// TIA Portal project "Reaktor2_Wizualizacja" (V17)

(* hardware
DEVICE "S7-1500/ET200MP station_1"  S7-1500 station
   slot 0: "Rail_0"  Rack  6ES7 590-1***0-0AA0
   slot 1: "PLC_1"  CPU 1512C-1 PN  6ES7 512-1CK00-0AB0  V2.9
      slot 3: "CPU display_1"  6ES7591-1AA00-0AA0
      slot 32768: "PROFINET interface_1"  X1
         slot 32769: "Port_1"  X1 P1
         slot 32770: "Port_2"  X1 P2
      slot 34817: "Virtual CP interface port_1"  Virtual CP interface port  Virtual CP interface port
DEVICE "PC_System_1"  SIMATIC PC station
   slot 0: "SIMATIC PC station"  Rail  SIMATIC PC-Station  V1.0
      slot 125: "Stationmanager"  Station_Manager  V6.0.4
   slot 1: "HMI_RT_1"  WinCC RT Professional  6AV2 105-0xxxx-xxxx  17.0.0.0
   slot 2: "IE general_1"  IE General  IE_CP  V8.2.0
      slot 1: "PROFINET interface"  IEGeneral.Interface.8.2.0
*)

// ===== PLC "PLC_1"  CPU 1512C-1 PN =====

VAR_GLOBAL   // PLC tag table "Default tag table"
   "System_Byte" AT %MB1 : Byte;
   "FirstScan" AT %M1.0 : Bool;
   "DiagStatusUpdate" AT %M1.1 : Bool;
   "AlwaysTRUE" AT %M1.2 : Bool;
   "AlwaysFALSE" AT %M1.3 : Bool;
   "Clock_Byte" AT %MB0 : Byte;
   "Clock_10Hz" AT %M0.0 : Bool;
   "Clock_5Hz" AT %M0.1 : Bool;
   "Clock_2.5Hz" AT %M0.2 : Bool;
   "Clock_2Hz" AT %M0.3 : Bool;
   "Clock_1.25Hz" AT %M0.4 : Bool;
   "Clock_1Hz" AT %M0.5 : Bool;
   "Clock_0.625Hz" AT %M0.6 : Bool;
   "Clock_0.5Hz" AT %M0.7 : Bool;
   "iAktualny_poziom" AT %MD8 : Real;   // czujnik pomiaru aktualnego poziomu czynników znajdujących się w reaktorze
   "iAktualna_temperatura" AT %MD12 : Real;   // czujnik pomiaru aktualnej wartości temperatury czynników znajdujących się w reaktorze
   "iWartość_zadana_poziomu" AT %MD16 : Real;   // AI3 - wartość zadana poziomu
   "iWartość_zadana_temperatury" AT %MD20 : Real;   // AI4 - wartość zadana temperatury
END_VAR

VAR_GLOBAL   // PLC tag table "zmienne_z_modułów"
   "xNapełnianie_reaktora" AT %M2.0 : Bool;   // Faza Napełnianie reaktora
   "xPodgrzewanie_produktu" AT %M2.1 : Bool;   // Faza Podgrzewanie produktu w reaktorze
   "xChłodzenie_reaktora" AT %M2.2 : Bool;   // Faza Chłodzenie produktu
   "xOpróżnianie_reaktora" AT %M2.3 : Bool;   // Faza Opróżnianie reaktora
   "xPraca_Man/Auto" AT %M2.4 : Bool;   // Przełącznik pracy Man/Auto
   "xZawór_V1" AT %M3.0 : Bool;   // zawór V1 - doprowadzenie czynnika A (oznaczenie V1)
   "xZawór_V2" AT %M3.1 : Bool;   // zawór V2 - doprowadzenie czynnika B (oznaczenie V2)
   "xZawór_V3" AT %M3.2 : Bool;   // Dopływ medium chłodzącego (oznaczenie V3)
   "xZawór_V4" AT %M3.3 : Bool;   // Odpływ medium chłodzącego (oznaczenie V4)
   "xZawór_V5" AT %M3.4 : Bool;   // V5 - Odpływ medium ogrzewającego (oznaczenie V5)
   "xSilnik_M" AT %M3.5 : Bool;   // M - Mieszadło wprawiane w ruch przez silnik (oznaczenie M)
   "iZawór_AV1" AT %MW4 : Int;   // Odprowadzenie produktu końcowego (oznaczenie AV1)
   "iZawór_AV2" AT %MW6 : Int;   // AV2 - Dopływ medium ogrzewającego (oznaczenie AV2)
END_VAR

DATA_BLOCK "Napełnianie_reaktora_DB"   // DB1
{ S7_Optimized_Access := 'FALSE' }
VERSION : 0.1
// stored: InstanceOfName Napełnianie_reaktora
"Napełnianie_reaktora"
BEGIN
END_DATA_BLOCK

DATA_BLOCK "Podgrzewanie_produktu_w_reaktorze_DB"   // DB2
{ S7_Optimized_Access := 'FALSE' }
VERSION : 0.1
// stored: InstanceOfName Podgrzewanie_produktu_w_reaktorze
"Podgrzewanie_produktu_w_reaktorze"
BEGIN
END_DATA_BLOCK

DATA_BLOCK "Chłodzenie_produktu_DB"   // DB3
{ S7_Optimized_Access := 'FALSE' }
VERSION : 0.1
// stored: InstanceOfName Chłodzenie_produktu
"Chłodzenie_produktu"
BEGIN
END_DATA_BLOCK

DATA_BLOCK "Opróżnianie_reaktora_DB"   // DB4
{ S7_Optimized_Access := 'FALSE' }
VERSION : 0.1
// stored: InstanceOfName Opróżnianie_reaktora
"Opróżnianie_reaktora"
BEGIN
END_DATA_BLOCK

DATA_BLOCK "zmienne_OB1"   // DB5
{ S7_Optimized_Access := 'FALSE' }
VERSION : 0.1
   VAR
      uiWybór_fazy_reaktora : UInt;
      iTemperatura_przed_podgrzaniem : Int;
      iNapełnianie_zbiornika_zakonczone : Int;
      iPodgrzewanie_produktu_zakończone : Int;
      iChłodzenie_reaktora_zakończone : Int;
      iOpróżnianie_reaktora_zakończone : Int;
      xAwaria : Bool;
      xZbocze_narastające_Napełnianie_zbiornika : Bool;
      xZbocze_narastające_Podgrzewanie_produktu : Bool;
      xZbocze_narastające_Chłodzenie_reaktora : Bool;
      xZbocze_narastające_Opróżnianie_reaktora : Bool;
   END_VAR
BEGIN
END_DATA_BLOCK

DATA_BLOCK "Użytkownicy"   // DB6
{ S7_Optimized_Access := 'TRUE' }
VERSION : 0.1
   VAR
      User_name : String;
   END_VAR
BEGIN
END_DATA_BLOCK

DATA_BLOCK "Symulator_grzanie_DB"   // DB8
{ S7_Optimized_Access := 'TRUE' }
VERSION : 0.1
// stored: InstanceOfName Symulator_grzanie
"Symulator_grzanie"
BEGIN
END_DATA_BLOCK

DATA_BLOCK "Symulator_napelniania_DB"   // DB11
{ S7_Optimized_Access := 'TRUE' }
VERSION : 0.1
// stored: InstanceOfName Symulator_napelniania
"Symulator_napelniania"
BEGIN
END_DATA_BLOCK

FUNCTION_BLOCK "Napełnianie_reaktora"   // FB1, SCL
{ S7_Optimized_Access := 'FALSE' }
VERSION : 0.1
   VAR_INPUT
      iAktualny_poziom_w_reaktorze : Real;
      iZadany_poziom : Real;
      iOpróżnianie_reaktora_zakończone : Int;
      xAwaria_lokal : Bool;
   END_VAR
   VAR_OUTPUT
      xZawór_V1 : Bool;   // zawór V1 - doprowadzenie czynnika A (oznaczenie V1)
      xZawór_V2 : Bool;   // zawór V2 - doprowadzenie czynnika B (oznaczenie V2)
      iNapełnianie_zbiornika_zakonczone : Int;
      iZawór_AV1 : Int;
   END_VAR
BEGIN
   ///zabezpiecznie że poprzednia faza opróżniania się zakończyła oraz nie wystąpiła awaria//////
   IF #xAwaria_lokal=0  THEN
       #iNapełnianie_zbiornika_zakonczone := 0;
       //napełnianie czynnikiem A do 1/3 poziomu zadanego otwarcie zaworu V1
       IF (#iAktualny_poziom_w_reaktorze >= 0.9 AND #iAktualny_poziom_w_reaktorze <= (#iZadany_poziom / 3.0)) THEN

           #xZawór_V1 := 1;

       END_IF;

       //po osiągnięciu 1/3 wartości zadanej zamknięcie zaworu V1, otwarcie zaworu V2
       IF (#iAktualny_poziom_w_reaktorze > (#iZadany_poziom / 3.0)) AND (#iAktualny_poziom_w_reaktorze <= #iZadany_poziom) THEN
           #xZawór_V1 := 0;
           #xZawór_V2 := 1;
       END_IF;

       //po osiągnięciu wartości zadanej zamknięcie zaworu V2
       IF (#iAktualny_poziom_w_reaktorze > #iZadany_poziom) THEN
           #xZawór_V2 := 0;
       END_IF;
       IF (#iAktualny_poziom_w_reaktorze > #iZadany_poziom) AND #xZawór_V2 = 0  THEN
           #iNapełnianie_zbiornika_zakonczone := 1;///informacja o zakończeniu fazy napełniania/////
       END_IF;
   END_IF;
   //wystąpienie awarii////
   IF #xAwaria_lokal=1 THEN
       ///zamknięcie zaworów V1, V2////
       #xZawór_V1 := 0;
       #xZawór_V2 := 0;
       ///otwarcie zaworu AV1 do opróżniania zbiornika/////
       IF #iAktualny_poziom_w_reaktorze > 0.0 THEN
           #iZawór_AV1 := 27648;

       END_IF;
       ///zamknięcie zaworu AV1 po opróżnieniu zbiornika////
       IF #iAktualny_poziom_w_reaktorze = 0.0 THEN
           #iZawór_AV1 := 0;
           #iNapełnianie_zbiornika_zakonczone := -1;///informacja o wystąpieniu awarii podczas napełniania////
       END_IF;

   END_IF;
END_FUNCTION_BLOCK

FUNCTION_BLOCK "Podgrzewanie_produktu_w_reaktorze"   // FB2, SCL
{ S7_Optimized_Access := 'FALSE' }
VERSION : 0.1
   VAR_INPUT
      iWartość_zadana_temperatury : Real;
      iAktualna_temperatura : Real;
      iNapełnianie_zbiornika_zakończone : Int;
      iAktualny_poziom_w_reaktorze : Real;
      xAwaria_lokalna : Bool;
   END_VAR
   VAR_OUTPUT
      xOdpływ_medium_ogrzewającego : Bool;
      xMieszadło : Bool;
      iDopływ_medium_ogrzewającego : Int;
      iTemperatura_przed_podgrzaniem : Real;
      iPodgrzewanie_produktu_zakończone : Int;
      iZawór_AV1 : Int;
   END_VAR
   VAR
      iI : Int := 0;
      iK : UInt := 0;
      iCzas_zamykania_zaworu_AV2 : UInt := 10;
      rWartość_zadana_temperatury : Real;
      rAktualna_temperatura : Real;
      rDopływ_medium_ogrzewającego : Real;
      xZbocze_narastające_1Hz : Bool;
   END_VAR
   VAR_TEMP
      "xStart_timera_zamykania zaworu" : Bool;
   END_VAR
BEGIN
   ///zabezpiecznie że poprzednia faza napełniania się zakończyła oraz nie wystąpiła awaria////// 
   IF #iNapełnianie_zbiornika_zakończone=1 AND #xAwaria_lokalna=0 THEN
       #iPodgrzewanie_produktu_zakończone := 0;


       //konwersja typów z INT na REAL
       #rAktualna_temperatura := INT_TO_REAL(#iAktualna_temperatura);
       #rWartość_zadana_temperatury := INT_TO_REAL(#iWartość_zadana_temperatury);

       //przepisanie temperatury produktu przed grzaniem
       WHILE #xOdpływ_medium_ogrzewającego = 0 AND #iI = 0 AND #rDopływ_medium_ogrzewającego <= 0.0 DO
           #iTemperatura_przed_podgrzaniem := #iAktualna_temperatura;
           #iI := #iI + 1;
           //Załączenie mieszadła 
           #xMieszadło := 1;
       END_WHILE;


       //otwarcie zaworu V5 odpływ medium ogrzewającego
       IF #xOdpływ_medium_ogrzewającego = 0 AND #iI = 1 THEN
           #xOdpływ_medium_ogrzewającego := 1;
       END_IF;

       //podgrzewanie produktu do 75% temperatury zadanej otwarcie zaworu AV2 - dopływ medium ogrzewającego
       IF (#rAktualna_temperatura <= (#rWartość_zadana_temperatury * 0.75)) AND (#xOdpływ_medium_ogrzewającego = 1) THEN
           #iDopływ_medium_ogrzewającego := 27648;
       END_IF;


       //po osiągnięciu 75% tempratury zadanej inicjalizacja zamkykania zaworu AV2 - dopływ medium ogrzewającego
       #rDopływ_medium_ogrzewającego := INT_TO_REAL(#iDopływ_medium_ogrzewającego);
       IF #rAktualna_temperatura >= (#rWartość_zadana_temperatury * 0.75) THEN

           #iDopływ_medium_ogrzewającego := 13500;

       END_IF;

       IF #rAktualna_temperatura >= #rWartość_zadana_temperatury THEN
           #iDopływ_medium_ogrzewającego := 0;
       END_IF;


           IF #iDopływ_medium_ogrzewającego<=0 THEN
               //Wyłącznie mieszadła
               #xMieszadło := 0;
               //zamknięcie zaworu V5 odpływ medium ogrzewającego
               #xOdpływ_medium_ogrzewającego := 0;
               #iPodgrzewanie_produktu_zakończone := 1;///informacja o zakończeniu fazy podgrzewania/////
           END_IF;

       END_IF;


   //wystąpienie awarii////
   IF #xAwaria_lokalna=1 THEN
       ///zamknięcie zaworów medium ogrzewającego oraz wyłączenie mieszadła////
       #iDopływ_medium_ogrzewającego := 0;
       #xOdpływ_medium_ogrzewającego := 0;
       #xMieszadło := 0;
       ///otwarcie zaworu AV1 do opróżniania zbiornika/////
       IF #iAktualny_poziom_w_reaktorze > 0.0 THEN
           #iZawór_AV1 := 27648;

       END_IF;
       ///zamknięcie zaworu AV1 po opróżnieniu zbiornika////
       IF #iAktualny_poziom_w_reaktorze = 0.0 THEN
           #iZawór_AV1 := 0;
           #iPodgrzewanie_produktu_zakończone := -1;///informacja o wystąpieniu awarii podczas fazy podgrzewania////
       END_IF;


   END_IF;
END_FUNCTION_BLOCK

FUNCTION_BLOCK "Chłodzenie_produktu"   // FB3, SCL
{ S7_Optimized_Access := 'FALSE' }
VERSION : 0.1
   VAR_INPUT
      iPodgrzewanie_produktu_zakończone : Int;
      iAktualna_temperatura : Real;
      iTemperatura_przed_podgrzaniem : Real;
      iAktualny_poziom_w_reaktorze : Real;
      xAwaria : Bool;
   END_VAR
   VAR_OUTPUT
      iChłodzenie_reaktora_zakończone : Int;
      xOdpływ_medium_chłodzącego : Bool;
      xDopływ_medium_chłodzącego : Bool;
      iZawór_AV1 : Int;
   END_VAR
BEGIN
   ///zabezpiecznie że poprzednia faza podgrzewania się zakończyła oraz nie wystąpiła awaria//////
   IF #iPodgrzewanie_produktu_zakończone = 1 AND #xAwaria = 0 THEN
       #iChłodzenie_reaktora_zakończone := 0;

       ///otwarcie zaworów medium chłodzącego
       IF #iChłodzenie_reaktora_zakończone = 0 AND #iAktualna_temperatura > #iTemperatura_przed_podgrzaniem THEN
           #xOdpływ_medium_chłodzącego := 1;
           #xDopływ_medium_chłodzącego := 1;
       ELSE
           ///zamknięcie zaworów medium chłodzącego////
           #xDopływ_medium_chłodzącego := 0;
           #xOdpływ_medium_chłodzącego := 0;
       END_IF;

       IF #iChłodzenie_reaktora_zakończone = 0 AND #iAktualna_temperatura <= #iTemperatura_przed_podgrzaniem THEN
           #iChłodzenie_reaktora_zakończone := 1;///informacja o zakończeniu fazy chłodzenia/////
       END_IF;

   END_IF;

   //wystąpienie awarii////
   IF #xAwaria=1 THEN
       ///zamknięcie zaworów medium chłodzącego////
       #xDopływ_medium_chłodzącego := 0;
       #xOdpływ_medium_chłodzącego := 0;
       ///otwarcie zaworu AV1 do opróżniania zbiornika/////
       IF #iAktualny_poziom_w_reaktorze > 0.0 THEN
           #iZawór_AV1 := 27648;

       END_IF;
       ///zamknięcie zaworu AV1 po opróżnieniu zbiornika////
       IF #iAktualny_poziom_w_reaktorze = 0.0 THEN
           #iZawór_AV1 := 0;
           #iChłodzenie_reaktora_zakończone := -1;///informacja o wystąpieniu awarii podczas fazy chłodzenia////
       END_IF;

   END_IF;
END_FUNCTION_BLOCK

FUNCTION_BLOCK "Opróżnianie_reaktora"   // FB4, SCL
{ S7_Optimized_Access := 'FALSE' }
VERSION : 0.1
   VAR_INPUT
      iChłodzenie_reaktora_zakończone : Int;
      iAktualny_poziom_w_reaktorze : Real;
      xAwaria_lokalna : Bool;
   END_VAR
   VAR_OUTPUT
      iOpróżnianie_reaktora_zakończone : Int;
      iZawór_AV1_odpływ : Int;
   END_VAR
BEGIN
   ///zabezpiecznie że poprzednia faza chłodzenia się zakończyła oraz nie wystąpiła awaria//////
   IF #iChłodzenie_reaktora_zakończone = 1 AND #xAwaria_lokalna= 0 THEN
       #iOpróżnianie_reaktora_zakończone := 0;

       ///otwarcie zaworu AV1 do opróżniania zbiornika/////
       IF #iOpróżnianie_reaktora_zakończone = 0 AND #iAktualny_poziom_w_reaktorze > 0 THEN
           #iZawór_AV1_odpływ := 27648;
       ELSE
           ///zamknięcie zaworu AV1 po opróżnieniu zbiornika////
           #iZawór_AV1_odpływ := 0;
       END_IF;

       IF #iOpróżnianie_reaktora_zakończone = 0 AND #iAktualny_poziom_w_reaktorze <= 1.0 THEN
           #iOpróżnianie_reaktora_zakończone := 1;///informacja o zakończeniu fazy opróżniania/////
       END_IF;

   END_IF;

   ///wystąpienie awarii////
   IF #iChłodzenie_reaktora_zakończone = 1 AND #xAwaria_lokalna = 1 THEN
       #iOpróżnianie_reaktora_zakończone := 0;

       ///otwarcie zaworu AV1 do opróżniania zbiornika/////
       IF #iOpróżnianie_reaktora_zakończone = 0 AND #iAktualny_poziom_w_reaktorze > 0 THEN
           #iZawór_AV1_odpływ := 27648;
       ELSE
           ///zamknięcie zaworu AV1 po opróżnieniu zbiornika////
           #iZawór_AV1_odpływ := 0;
       END_IF;

       IF #iOpróżnianie_reaktora_zakończone = 0 AND #iAktualny_poziom_w_reaktorze <= 1.0 THEN
           #iOpróżnianie_reaktora_zakończone := -1;///informacja o wystąpieniu awarii podczas fazy opróżniania////
       END_IF;

   END_IF;
END_FUNCTION_BLOCK

FUNCTION_BLOCK "Symulator_napelniania"   // FB5, SCL
{ S7_Optimized_Access := 'TRUE' }
VERSION : 0.1
   VAR_INPUT
      iZadany_poziom : Int;
      xZawór_V1 : Bool;
      xZawór_V2 : Bool;
      iZawór_AV1 : Int;
   END_VAR
   VAR_IN_OUT
      dAktualny_poziom_w_reaktorze : Real;
   END_VAR
   VAR
      ddAktualny_poziom_w_reaktorze : Real;
   END_VAR
   VAR CONSTANT
      h : Real := 0.1;
   END_VAR
BEGIN
   IF #xZawór_V1 = 1 OR #xZawór_V2 = 1 AND #iZawór_AV1 = 0 AND #dAktualny_poziom_w_reaktorze < 13.0  THEN
       #ddAktualny_poziom_w_reaktorze := 0.125;
       #dAktualny_poziom_w_reaktorze := #dAktualny_poziom_w_reaktorze + #ddAktualny_poziom_w_reaktorze * #h;
   END_IF;


   IF #xZawór_V1 = 0 AND #xZawór_V2 = 0 AND #iZawór_AV1 > 0 AND #dAktualny_poziom_w_reaktorze > 1.0 THEN
       #ddAktualny_poziom_w_reaktorze := (INT_TO_REAL(#iZawór_AV1) / 27648) * 0.175 * #dAktualny_poziom_w_reaktorze;
       #dAktualny_poziom_w_reaktorze := #dAktualny_poziom_w_reaktorze - #ddAktualny_poziom_w_reaktorze * #h;
   END_IF;
END_FUNCTION_BLOCK

FUNCTION_BLOCK "Block_1"   // FB6, SCL
{ S7_Optimized_Access := 'TRUE' }
VERSION : 0.1
   VAR_INPUT
      xNapełnianie : Bool;
      xPodgrzewanie : Bool;
      xChłodzenie : Bool;
      xOpróżnianie : Bool;
   END_VAR
   VAR_OUTPUT
      uiFaza_reaktora : UInt;
   END_VAR
BEGIN

   IF #xNapełnianie = 1 THEN
       #uiFaza_reaktora := 1;

   ELSIF #xPodgrzewanie = 1 THEN
       #uiFaza_reaktora := 2;

   ELSIF #xChłodzenie = 1 THEN
       #uiFaza_reaktora := 3;

   ELSIF #xOpróżnianie = 1 THEN
       #uiFaza_reaktora := 4;

   END_IF;
END_FUNCTION_BLOCK

FUNCTION_BLOCK "Symulator_grzanie"   // FB7, SCL
{ S7_Optimized_Access := 'TRUE' }
VERSION : 0.1
   VAR_INPUT
      wysokość : Real;
      iZawór_AV2 : Int;
      xZawór_V3 : Bool;
   END_VAR
   VAR_IN_OUT
      Temp_w_zbiorniku : Real;
   END_VAR
   VAR_TEMP
      Temp_w_wymienniku : Real;
      dd_temp_w_zbiorniku : Real;
      F : Real;
      V : Real;
   END_VAR
   VAR CONSTANT
      k : Real := 10000.0;
      cw : Real := 4200.0;
      ro : Real := 1.0;
      pp : Real := 20.0;
      h : Real := 0.1;
   END_VAR
BEGIN
   IF #iZawór_AV2 > 0 THEN
       #Temp_w_wymienniku := 150;
       #F := INT_TO_REAL(#iZawór_AV2) / 27648 * 0.9;
       #V := #pp * #wysokość;
       #dd_temp_w_zbiorniku := ((#k * #F) / (#cw * #ro * #V)) * (#Temp_w_wymienniku - #Temp_w_zbiorniku);
       #Temp_w_zbiorniku := #Temp_w_zbiorniku + #dd_temp_w_zbiorniku * #h;
   END_IF;

   IF #xZawór_V3 =1 THEN
       #Temp_w_wymienniku := 14 ;
       #F := 2;
       #V := #pp * #wysokość;
       #dd_temp_w_zbiorniku := ((#k * #F) / (#cw * #ro * #V)) * (#Temp_w_zbiorniku - #Temp_w_wymienniku);
       #Temp_w_zbiorniku := #Temp_w_zbiorniku - #dd_temp_w_zbiorniku * #h;
   END_IF;
END_FUNCTION_BLOCK

FUNCTION "FC_wybór_fazy_reaktora" : Void   // FC1, SCL
{ S7_Optimized_Access := 'TRUE' }
VERSION : 0.1
   VAR_INPUT
      xNapełnianie : Bool;
      xPodgrzewanie : Bool;
      xChłodzenie : Bool;
      xOpróżnianie : Bool;
   END_VAR
   VAR_IN_OUT
      uiFaza_reaktora_1 : UInt;
   END_VAR
BEGIN

   IF #xNapełnianie=1 OR #uiFaza_reaktora_1 = 1 THEN
       #uiFaza_reaktora_1 := 1;

   ELSIF #xPodgrzewanie=1 OR #uiFaza_reaktora_1 = 2  THEN
       #uiFaza_reaktora_1 := 2;

   ELSIF #xChłodzenie=1 OR #uiFaza_reaktora_1 = 3 THEN
       #uiFaza_reaktora_1 := 3;

   ELSIF #xOpróżnianie=1 OR #uiFaza_reaktora_1 = 4 THEN
       #uiFaza_reaktora_1 := 4;

   END_IF;
END_FUNCTION

ORGANIZATION_BLOCK "Main"   // OB1, SCL, ProgramCycle
TITLE = "Main Program Sweep (Cycle)"
{ S7_Optimized_Access := 'TRUE' }
VERSION : 0.1
   VAR_INPUT
      Initial_Call : Bool;   // Initial call of this OB
      Remanence : Bool;   // =True, if remanent data are available
   END_VAR
BEGIN
   IF "FirstScan" = 1 THEN
       "iAktualna_temperatura" := 20.0;
       "iAktualny_poziom" := 1.0
       ;
   END_IF;


   //"R_TRIG_DB_1"(CLK := "xNapełnianie_reaktora",
                 //Q => "zmienne_OB1".xZbocze_narastające_Napełnianie_zbiornika);

   ///wybór fazy procesu oraz przypisanie jej odpowiedniego numeru////
   "FC_wybór_fazy_reaktora"(xNapełnianie := "xNapełnianie_reaktora",
                            xPodgrzewanie := "xPodgrzewanie_produktu",
                            xChłodzenie := "xChłodzenie_reaktora",
                            xOpróżnianie := "xOpróżnianie_reaktora",
                            uiFaza_reaktora_1:="zmienne_OB1".uiWybór_fazy_reaktora);



   ////uruchamianie odpowiedniej fazy procesu zgodnie z przypisanym numerem////
   CASE "zmienne_OB1".uiWybór_fazy_reaktora OF
       1:
           "Napełnianie_reaktora_DB"(iAktualny_poziom_w_reaktorze := "iAktualny_poziom",
                                     iZadany_poziom := "iWartość_zadana_poziomu",
                                     iOpróżnianie_reaktora_zakończone := "zmienne_OB1".iOpróżnianie_reaktora_zakończone,
                                     xZawór_V1 => "xZawór_V1",
                                     xZawór_V2 => "xZawór_V2",
                                     iZawór_AV1 => "iZawór_AV1",
                                     iNapełnianie_zbiornika_zakonczone => "zmienne_OB1".iNapełnianie_zbiornika_zakonczone);

           IF "xPraca_Man/Auto" = 0 AND "xPodgrzewanie_produktu" = 1 AND "zmienne_OB1".iNapełnianie_zbiornika_zakonczone = 1 THEN
               "zmienne_OB1".uiWybór_fazy_reaktora := 2;
           END_IF;
           IF "xPraca_Man/Auto" = 1 AND "zmienne_OB1".iNapełnianie_zbiornika_zakonczone = 1 THEN
               "zmienne_OB1".uiWybór_fazy_reaktora := 2;
           END_IF;
           IF "zmienne_OB1".iNapełnianie_zbiornika_zakonczone = -1 THEN
               "zmienne_OB1".uiWybór_fazy_reaktora := 5;
           END_IF;



       2:
           "Podgrzewanie_produktu_w_reaktorze_DB"(iWartość_zadana_temperatury := "iWartość_zadana_temperatury",
                                                  iAktualna_temperatura := "iAktualna_temperatura",
                                                  iAktualny_poziom_w_reaktorze := "iAktualny_poziom",
                                                  xAwaria_lokalna := "zmienne_OB1".xAwaria,
                                                  iNapełnianie_zbiornika_zakończone := "zmienne_OB1".iNapełnianie_zbiornika_zakonczone,
                                                  xOdpływ_medium_ogrzewającego => "xZawór_V5",
                                                  xMieszadło => "xSilnik_M",
                                                  iDopływ_medium_ogrzewającego => "iZawór_AV2",
                                                  iZawór_AV1 => "iZawór_AV1",
                                                  iTemperatura_przed_podgrzaniem => "zmienne_OB1".iTemperatura_przed_podgrzaniem,
                                                  iPodgrzewanie_produktu_zakończone => "zmienne_OB1".iPodgrzewanie_produktu_zakończone);

           IF "xPraca_Man/Auto" = 0 AND "xChłodzenie_reaktora" = 1 AND "zmienne_OB1".iPodgrzewanie_produktu_zakończone = 1 THEN
               "zmienne_OB1".uiWybór_fazy_reaktora := 3;
           END_IF;
           IF "xPraca_Man/Auto" = 1 AND "zmienne_OB1".iPodgrzewanie_produktu_zakończone = 1 THEN
               "zmienne_OB1".uiWybór_fazy_reaktora := 3;
           END_IF;
           IF "zmienne_OB1".iPodgrzewanie_produktu_zakończone = -1 THEN
               "zmienne_OB1".uiWybór_fazy_reaktora := 5;
           END_IF;

       3:
           "Chłodzenie_produktu_DB"(iPodgrzewanie_produktu_zakończone := "zmienne_OB1".iPodgrzewanie_produktu_zakończone,
                                    iAktualna_temperatura := "iAktualna_temperatura",
                                    iAktualny_poziom_w_reaktorze := "iAktualny_poziom",
                                    xAwaria := "zmienne_OB1".xAwaria,
                                    iTemperatura_przed_podgrzaniem := "zmienne_OB1".iTemperatura_przed_podgrzaniem,
                                    iChłodzenie_reaktora_zakończone => "zmienne_OB1".iChłodzenie_reaktora_zakończone,
                                    xDopływ_medium_chłodzącego => "xZawór_V3",
                                    xOdpływ_medium_chłodzącego => "xZawór_V4",
                                    iZawór_AV1 => "iZawór_AV1");

           IF "xPraca_Man/Auto" = 0 AND "xOpróżnianie_reaktora" = 1 AND "zmienne_OB1".iChłodzenie_reaktora_zakończone = 1 THEN
               "zmienne_OB1".uiWybór_fazy_reaktora := 4;
           END_IF;
           IF "xPraca_Man/Auto" = 1 AND "zmienne_OB1".iChłodzenie_reaktora_zakończone = 1 THEN
               "zmienne_OB1".uiWybór_fazy_reaktora := 4;
           END_IF;
           IF "zmienne_OB1".iChłodzenie_reaktora_zakończone = -1 THEN
               "zmienne_OB1".uiWybór_fazy_reaktora := 5;
           END_IF;
       4:
           "Opróżnianie_reaktora_DB"(iChłodzenie_reaktora_zakończone := "zmienne_OB1".iChłodzenie_reaktora_zakończone,
                                     iAktualny_poziom_w_reaktorze := "iAktualny_poziom",
                                     xAwaria_lokalna := "zmienne_OB1".xAwaria,
                                     iOpróżnianie_reaktora_zakończone => "zmienne_OB1".iOpróżnianie_reaktora_zakończone,
                                     iZawór_AV1_odpływ => "iZawór_AV1");

           IF "zmienne_OB1".iOpróżnianie_reaktora_zakończone = 1 THEN
               "zmienne_OB1".uiWybór_fazy_reaktora := 5;
           END_IF;
           IF "zmienne_OB1".iOpróżnianie_reaktora_zakończone = -1 THEN
               "zmienne_OB1".uiWybór_fazy_reaktora := 5;
           END_IF;


            ELSE
            IF "xPraca_Man/Auto" = 0 AND "xNapełnianie_reaktora" = 1 AND "zmienne_OB1".xAwaria = 0 THEN
              "zmienne_OB1".uiWybór_fazy_reaktora := 1;
            END_IF;
           IF "xPraca_Man/Auto" = 1 AND "zmienne_OB1".xAwaria = 0 THEN
            "zmienne_OB1".uiWybór_fazy_reaktora := 1;
            END_IF;

           ///wystąpienie awarii////
           IF "zmienne_OB1".xAwaria = 1 THEN
               "zmienne_OB1".iNapełnianie_zbiornika_zakonczone := 0;
               "zmienne_OB1".iPodgrzewanie_produktu_zakończone := 0;
               "zmienne_OB1".iChłodzenie_reaktora_zakończone := 0;
               "zmienne_OB1".iOpróżnianie_reaktora_zakończone := 0;
           END_IF;
   END_CASE;
END_ORGANIZATION_BLOCK

ORGANIZATION_BLOCK "Symulator"   // OB30, SCL, CyclicInterrupt
{ S7_Optimized_Access := 'TRUE' }
VERSION : 0.1
   VAR_INPUT
      Initial_Call : Bool;   // Initial call of this OB
      Event_Count : Int;   // Events discarded
   END_VAR
BEGIN




   "Symulator_napelniania_DB"(iZadany_poziom := "iWartość_zadana_poziomu",
                              xZawór_V1 := "xZawór_V1",
                              xZawór_V2 := "xZawór_V2",
                              iZawór_AV1 := "iZawór_AV1",
                              dAktualny_poziom_w_reaktorze := "iAktualny_poziom");

   "Symulator_grzanie_DB"(wysokość:="iAktualny_poziom",
                          iZawór_AV2:="iZawór_AV2",
                          xZawór_V3:="xZawór_V3",
                          Temp_w_zbiorniku:="iAktualna_temperatura");
END_ORGANIZATION_BLOCK

(* ===== HMI "HMI_RT_1" =====
system functions are stored by id; their names below are inferred from use
connection "HMI_Connection_1": S71200_TCP_IP, SCADA_S7_1500_OMS

HMI tags "Default tag table"
   "Napełnianie_reaktora_DB_iZadany_poziom" : Real = PLC Napełnianie_reaktora_DB.iZadany_poziom AT %DB1.DBD4, 500 ms
   "xNapełnianie_reaktora" : Bool = PLC xNapełnianie_reaktora AT %M2.0, 500 ms
   "xPodgrzewanie_produktu" : Bool = PLC xPodgrzewanie_produktu AT %M2.1, 500 ms
   "xChłodzenie_reaktora" : Bool = PLC xChłodzenie_reaktora AT %M2.2, 500 ms
   "xOpróżnianie_reaktora" : Bool = PLC xOpróżnianie_reaktora AT %M2.3, 500 ms
   "Napełnianie_reaktora_DB_iNapełnianie_zbiornika_zakonczone" : Int = PLC Napełnianie_reaktora_DB.iNapełnianie_zbiornika_zakonczone AT %DB1.DBW14, 500 ms
   "Podgrzewanie_produktu_w_reaktorze_DB_iPodgrzewanie_produktu_zakończone" : Int = PLC Podgrzewanie_produktu_w_reaktorze_DB.iPodgrzewanie_produktu_zakończone AT %DB2.DBW24, 500 ms
   "Chłodzenie_produktu_DB_iChłodzenie_reaktora_zakończone" : Int = PLC Chłodzenie_produktu_DB.iChłodzenie_reaktora_zakończone AT %DB3.DBW16, 500 ms
   "Opróżnianie_reaktora_DB_iOpróżnianie_reaktora_zakończone" : Int = PLC Opróżnianie_reaktora_DB.iOpróżnianie_reaktora_zakończone AT %DB4.DBW8, 500 ms
   "Napełnianie_reaktora_DB_iAktualny_poziom_w_reaktorze" : Real = PLC Napełnianie_reaktora_DB.iAktualny_poziom_w_reaktorze AT %DB1.DBD0, 500 ms
   "Podgrzewanie_produktu_w_reaktorze_DB_xMieszadło" : Bool = PLC Podgrzewanie_produktu_w_reaktorze_DB.xMieszadło AT %DB2.DBX16.1, 500 ms
   "xPraca_Man/Auto" : Bool = PLC "xPraca_Man/Auto" AT %M2.4, 500 ms
   "Podgrzewanie_produktu_w_reaktorze_DB_iAktualna_temperatura" : Real = PLC Podgrzewanie_produktu_w_reaktorze_DB.iAktualna_temperatura AT %DB2.DBD4, 500 ms
   "Podgrzewanie_produktu_w_reaktorze_DB_iWartość_zadana_temperatury" : Real = PLC Podgrzewanie_produktu_w_reaktorze_DB.iWartość_zadana_temperatury AT %DB2.DBD0, 500 ms
   "xZawór_V1" : Bool = PLC xZawór_V1 AT %M3.0, 500 ms
   "xZawór_V2" : Bool = PLC xZawór_V2 AT %M3.1, 500 ms
   "xZawór_V3" : Bool = PLC xZawór_V3 AT %M3.2, 500 ms
   "xZawór_V4" : Bool = PLC xZawór_V4 AT %M3.3, 500 ms
   "xZawór_V5" : Bool = PLC xZawór_V5 AT %M3.4, 500 ms
   "iZawór_AV1" : Int = PLC iZawór_AV1 AT %MW4, 500 ms
   "Opróżnianie_reaktora_DB_iZawór_AV1_odpływ" : Int = PLC Opróżnianie_reaktora_DB.iZawór_AV1_odpływ AT %DB4.DBW10, 500 ms
   "Podgrzewanie_produktu_w_reaktorze_DB_iDopływ_medium_ogrzewającego" : Int = PLC Podgrzewanie_produktu_w_reaktorze_DB.iDopływ_medium_ogrzewającego AT %DB2.DBW18, 500 ms
   "Chłodzenie_produktu_DB_xDopływ_medium_chłodzącego" : Bool = PLC Chłodzenie_produktu_DB.xDopływ_medium_chłodzącego AT %DB3.DBX18.1, 500 ms
   "Chłodzenie_produktu_DB_xOdpływ_medium_chłodzącego" : Bool = PLC Chłodzenie_produktu_DB.xOdpływ_medium_chłodzącego AT %DB3.DBX18.0, 500 ms
   "Podgrzewanie_produktu_w_reaktorze_DB_xOdpływ_medium_ogrzewającego" : Bool = PLC Podgrzewanie_produktu_w_reaktorze_DB.xOdpływ_medium_ogrzewającego AT %DB2.DBX16.0, 500 ms
   "iZawór_AV2" : Int = PLC iZawór_AV2 AT %MW6, 500 ms
   "iAktualny_poziom" : Real = PLC iAktualny_poziom AT %MD8, 500 ms
   "iAktualna_temperatura" : Real = PLC iAktualna_temperatura AT %MD12, 500 ms
   "User_name" : String[254] = PLC Użytkownicy.User_name AT %DB1.DBX0.0, 500 ms

screen "Screen_1" 1024x768
   Group "Group" at 375,155 size 159x196
   Group "Group_2" at 347,181 size 214x211
   EllipticalArc "Elliptical arc_1" at 216,469 size 24x11
   Polygon "Polygon_2" at 265,373 size 24x20
      Appearance <- "xZawór_V1"
   Polygon "Polygon_3" at 265,353 size 24x20
      Appearance <- "xZawór_V1"
   Group "Group_7" at 265,353 size 24x40
   Group "Group_6" at 215,361 size 60x20
   EllipticalArc "Elliptical arc_2" at 301,528 size 24x11
   Polygon "Polygon_4" at 353,423 size 24x20
      Appearance <- "xZawór_V5"
   Polygon "Polygon_5" at 353,403 size 24x20
      Appearance <- "xZawór_V5"
   EllipticalArc "Elliptical arc_3" at 678,469 size 24x11
   Polygon "Polygon_1" at 629,373 size 24x20
      Appearance <- "xZawór_V2"
   Polygon "Polygon_6" at 629,353 size 24x20
      Appearance <- "xZawór_V2"
   Group "Group_13" at 629,353 size 24x40
   Group "Group_14" at 643,361 size 60x20
   RoundButton "Round button_1" at 856,110 size 40x40; Text 'Text'
      on PressLeft: SetBit("xNapełnianie_reaktora")
      on ReleaseLeft: ResetBit("xNapełnianie_reaktora")
   RoundButton "Round button_2" at 856,168 size 40x40; Text 'Text'
      on PressLeft: SetBit("xPodgrzewanie_produktu")
      on ReleaseLeft: ResetBit("xPodgrzewanie_produktu")
   RoundButton "Round button_3" at 856,225 size 40x40; Text 'Text'
      on PressLeft: SetBit("xChłodzenie_reaktora")
      on ReleaseLeft: ResetBit("xChłodzenie_reaktora")
   RoundButton "Round button_4" at 856,283 size 40x40; Text 'Text'
      on PressLeft: SetBit("xOpróżnianie_reaktora")
      on ReleaseLeft: ResetBit("xOpróżnianie_reaktora")
   RoundButton "Round button_5" at 856,437 size 48x48; Text 'Text'
      on PressLeft: ResetBit("xPraca_Man/Auto")
      on ReleaseLeft: ResetBit("xPraca_Man/Auto")
   RoundButton "Round button_6" at 856,355 size 48x48; Text 'Text'
      on PressLeft: SetBit("xPraca_Man/Auto")
      on ReleaseLeft: SetBit("xPraca_Man/Auto")
   TextField "Text field_8" at 859,406 size 46x23; Text 'AUTO'
   TextField "Text field_9" at 861,489 size 40x23; Text 'CYKL'
   EllipticalArc "Elliptical arc_4" at 189,111 size 11x24
   TextField "Text field_16" at 443,109 size 26x25; Text '3~'
   Rectangle "Rectangle_8" at 451,328 size 9x12
      Appearance <- "Podgrzewanie_produktu_w_reaktorze_DB_xMieszadło"
   Rectangle "Rectangle_9" at 432,318 size 12x9
      Appearance <- "Podgrzewanie_produktu_w_reaktorze_DB_xMieszadło"
   Rectangle "Rectangle_10" at 466,318 size 12x9
      Appearance <- "Podgrzewanie_produktu_w_reaktorze_DB_xMieszadło"
   Rectangle "Rectangle_11" at 451,303 size 9x12
      Appearance <- "Podgrzewanie_produktu_w_reaktorze_DB_xMieszadło"
   EllipticalArc "Elliptical arc_5" at 767,142 size 11x24
   Polygon "Polygon_7" at 671,191 size 20x24
      Appearance <- "xZawór_V3"
   Polygon "Polygon_8" at 651,191 size 20x24
      Appearance <- "xZawór_V3"
   Group "Group_25" at 651,191 size 40x24
   Group "Group_29" at 131,142 size 77x24
   TextField "Text field_19" at 87,141 size 39x27; Text 'AV2'
   Group "Group_3" at 347,181 size 214x211
   Group "Group_1" at 375,155 size 159x196
   WindowSlider "Scroll bar_1" at 216,273 size 21x62; Authorization "Monitor"
      ProcessValue <- "Napełnianie_reaktora_DB_iZadany_poziom"
   IOField "I/O field_1" at 135,246 size 80x20; FormatPattern s999999999.999
      ProcessValue <- "Napełnianie_reaktora_DB_iZadany_poziom"
   TextField "Text field_4" at 886,89 size 13x21; Text 'N'
   TextField "Text field_5" at 886,151 size 13x21; Text 'G'
   TextField "Text field_6" at 886,207 size 12x21; Text 'C'
   TextField "Text field_7" at 886,265 size 14x21; Text 'O'
   Group "Group_18" at 365,111 size 60x20
   Group "Group_17" at 435,101 size 40x40
   Group "Group_16" at 189,111 size 167x24
   TextField "Text field_17" at 160,111 size 17x25; Text 'M'
   Bar "Bar_2" at 417,181 size 78x120; MinimumValue 0; MaximumValue 12
      ProcessValue <- "iAktualny_poziom"
   Group "Group_19" at 856,110 size 40x213; Authorization "Monitor"
   Group "Group_20" at 432,303 size 46x37
   Group "Group_21" at 432,303 size 46x37
   GraphicView "Graphic view_6" at 703,166 size 75x75; Picture "Graphic_13"
   GraphicView "Graphic view_4" at 127,166 size 75x75; Picture "Graphic_14"
   GraphicView "Graphic view_7" at 507,465 size 75x75; Picture "Graphic_3"
   Group "Group_34" at 585,462 size 24x77
   TextField "Text field_20" at 585,550 size 26x27; Text 'V4'
   Group "Group_35" at 533,403 size 24x40
   Group "Group_36" at 547,411 size 60x20
   TextField "Text field_21" at 442,568 size 39x27; Text 'AV1'
   WindowSlider "Scroll bar_2" at 682,273 size 21x62; Authorization "Monitor"
      ProcessValue <- "Podgrzewanie_produktu_w_reaktorze_DB_iWartość_zadana_temperatury"
   IOField "I/O field_2" at 704,246 size 80x20; FormatPattern s999999999.999
      ProcessValue <- "Podgrzewanie_produktu_w_reaktorze_DB_iWartość_zadana_temperatury"
   Bar "Bar_1" at 502,181 size 20x120; MinimumValue 0; MaximumValue 12
      ProcessValue <- "iAktualna_temperatura"
   TextField "Text field_22" at 237,337 size 28x16; Text 'Hzad'
   TextField "Text field_23" at 654,336 size 28x16; Text 'Tzad'
   Circle "Circle_17" at 564,235 size 16x16
      Appearance <- "xNapełnianie_reaktora"
   Circle "Circle_18" at 564,265 size 16x16
      Appearance <- "xPodgrzewanie_produktu"
   Circle "Circle_19" at 564,295 size 16x16
      Appearance <- "xChłodzenie_reaktora"
   Circle "Circle_20" at 564,325 size 16x16
      Appearance <- "xOpróżnianie_reaktora"
   Circle "Circle_21" at 564,355 size 16x16
      Appearance <- "xPraca_Man/Auto"
   Circle "Circle_22" at 564,385 size 16x16
      Appearance <- "xPraca_Man/Auto"
   TextField "Text field_10" at 580,236 size 10x18; Text 'N'
   TextField "Text field_11" at 581,266 size 10x18; Text 'G'
   TextField "Text field_12" at 580,296 size 10x18; Text 'C'
   TextField "Text field_13" at 581,325 size 11x18; Text 'O'
   TextField "Text field_14" at 582,354 size 35x18; Text 'AUTO'
   TextField "Text field_15" at 581,385 size 30x18; Text 'CYKL'
   GraphicView "Graphic view_3" at 240,413 size 75x75; Picture "Graphic_4"
   Group "Group_5" at 216,403 size 24x77
   TextField "Text field_1" at 215,488 size 26x27; Text 'V1'
   Group "Group_4" at 215,353 size 74x40
   GraphicView "Graphic view_1" at 603,413 size 75x75; Picture "Graphic_4"
   Group "Group_12" at 678,403 size 24x77
   TextField "Text field_3" at 677,488 size 26x27; Text 'V2'
   Group "Group_15" at 629,353 size 74x40
   Group "Group_24" at 701,142 size 77x24
   TextField "Text field_18" at 786,141 size 26x27; Text 'V3'
   GraphicView "Graphic view_2" at 328,465 size 75x75; Picture "Graphic_3"
   Group "Group_9" at 301,462 size 24x77
   TextField "Text field_2" at 299,550 size 26x27; Text 'V5'
   Group "Group_10" at 353,403 size 24x40
   Group "Group_11" at 303,411 size 60x20
   Group "Group_37" at 439,427 size 39x46
   GraphicView "Graphic view_8" at 420,500 size 75x75; Picture "Graphic_3"
   Group "Group_8" at 651,144 size 40x71
   Group "Group_22" at 218,144 size 40x71
   Group "Group_23" at 856,355 size 49x157; Authorization "Operate"
   EllipticalArc "Elliptical arc_6" at 131,142 size 11x24
   Polygon "Polygon_9" at 218,191 size 20x24
      Appearance <- "iZawór_AV2"
   Polygon "Polygon_10" at 238,191 size 20x24
      Appearance <- "iZawór_AV2"
   Group "Group_30" at 218,191 size 40x24
   EllipticalArc "Elliptical arc_7" at 585,528 size 24x11
   Polygon "Polygon_11" at 533,423 size 24x20
      Appearance <- "xZawór_V4"
   Polygon "Polygon_12" at 533,403 size 24x20
      Appearance <- "xZawór_V4"
   Polygon "Polygon_13" at 439,450 size 39x23
      Appearance <- "iZawór_AV1"
   Polygon "Polygon_14" at 439,427 size 39x23
      Appearance <- "iZawór_AV1"

screen "User_Admin" 1024x768
   UserView "User view_1" at 116,151 size 579x192
   TextField "Text field_1" at 213,69 size 415x60; Text 'User Administration'
   Button "Button_1" at 615,369 size 80x30; TextOff 'Login'
      on ReleaseLeft: function_a2a04561()
   TextField "Text field_24" at 160,378 size 107x21; Text 'Logged user:'
   IOField "I/O field_1" at 307,379 size 145x20; FormatPattern AAAA
      ProcessValue <- "User_name"
*)